// TIA Portal V20 export
DATA_BLOCK "CallEquipment_DB"   // DB155
{ DB_Accessible_From_OPC_UA := 'FALSE' }
// stored: AssignedProDiagFB Unit1.Em2.ProDiag, DBAccessibleFromOPCUA false, DBAccessibleFromWebserver false, InstanceOfName Unit1.Em2.CallEquipment, InstanceOfType FB, Namespace Unit1.Em2
"Unit1.Em2.CallEquipment"
   // VAR_INPUT
   //    ZoneOperationEnable { ExternalWritable := 'False'} : "LWONIK_typeSafetyZoneManualOperation";
   //    unitEnableControlInterfaces { ExternalWritable := 'False'} : "LAF_typeEnableControlInterfaces";
   //    commandExcute { ExternalWritable := 'False'} : Bool;
   // END_VAR
   // VAR_IN_OUT
   //    unitStatus : "LAF_typeUnitStatus";
   //    emFeedback : "LUC_typeEmFeedback";
   //    unitAlarmDB : "LAF_typeAlarms";
   // END_VAR
   // VAR
   //    instSequenceSemiAutoSplice { ExternalWritable := 'False'} : "Unit1.Em2.Sequence_1_SemiAutoSplice";
   //    instTapeUnitInitializedJob1 { ExternalWritable := 'False'} : "LAF_SelectJob";
   //    instAutoSplicerModuleInitializedJob2 { ExternalWritable := 'False'} : "LAF_SelectJob";
   //    instLeftSplicingModuleMoverInitializedJob3 { ExternalWritable := 'False'} : "LAF_SelectJob";
   //    instRightSplicingModuleMoverInitializedJob4 { ExternalWritable := 'False'} : "LAF_SelectJob";
   //    instSplicingModuleMoverAutoJob5 { ExternalWritable := 'False'} : "LAF_SelectJob";
   //    instVacuumAutoJob7 { ExternalWritable := 'False'} : "LAF_SelectJob";
   //    instCutterAutoJob8 { ExternalWritable := 'False'} : "LAF_SelectJob";
   //    instLeftElectrodeReMoverAutoJob9 { ExternalWritable := 'False'} : "LAF_SelectJob";
   //    instRightElectrodeReMoverAutoJob10 { ExternalWritable := 'False'} : "LAF_SelectJob";
   //    instTapeAttachReadyAutoJob11 { ExternalWritable := 'False'} : "LAF_SelectJob";
   //    instTapeAttachStartAutoJob12 { ExternalWritable := 'False'} : "LAF_SelectJob";
   //    instTapeAttachFinishAutoJob13 { ExternalWritable := 'False'} : "LAF_SelectJob";
   //    instLeftSplicingModuleMoverAutoJob14 { ExternalWritable := 'False'} : "LAF_SelectJob";
   //    instRightSplicingModuleMoverAutoJob15 { ExternalWritable := 'False'} : "LAF_SelectJob";
   //    instSemiAutoSpliceFullAutoJob20 { ExternalWritable := 'False'} : "LAF_SelectJob";
   //    instElectrodeFixRightTopFwdBwd { ExternalWritable := 'False'} : "LBC_TwoWayActuatorCn";
   //    instElectrodeFixRightBottomFwdBwd { ExternalWritable := 'False'} : "LBC_TwoWayActuatorCn";
   //    instElectrodeFixLeftTopFwdBwd { ExternalWritable := 'False'} : "LBC_TwoWayActuatorCn";
   //    instElectrodeFixLeftBottomFwdBwd { ExternalWritable := 'False'} : "LBC_TwoWayActuatorCn";
   //    instElectrodeFixLeftTopUpDown { ExternalWritable := 'False'} : "LBC_TwoWayActuatorCn";
   //    instElectrodeFixLeftBottomUpDown { ExternalWritable := 'False'} : "LBC_TwoWayActuatorCn";
   //    instUwSemiSplicerVacuumRightTopOnOff { ExternalWritable := 'False'} : "LBC_TwoWayActuatorCn";
   //    instUwSemiSplicerVacuumRightBottomOnOff { ExternalWritable := 'False'} : "LBC_TwoWayActuatorCn";
   //    instUwSemiSplicerVacuumLeftTopOnOff { ExternalWritable := 'False'} : "LBC_TwoWayActuatorCn";
   //    instUwSemiSplicerVacuumLeftBottomOnOff { ExternalWritable := 'False'} : "LBC_TwoWayActuatorCn";
   //    instElectrodeCutterFwdBwd { ExternalWritable := 'False'} : "LBC_TwoWayActuatorCn";
   //    instSplicingLeftModuleMoverFwdBwd { ExternalWritable := 'False'} : "LBC_TwoWayActuatorCn";
   //    instSplicingRightModuleMoverFwdBwd { ExternalWritable := 'False'} : "LBC_TwoWayActuatorCn";
   //    instElectrodeLeftHolderMoverFwdBwd { ExternalWritable := 'False'} : "LBC_TwoWayActuatorCn";
   //    instElectrodeRightHolderMoverFwdBwd { ExternalWritable := 'False'} : "LBC_TwoWayActuatorCn";
   //    instTapeLoadingTurnCwCcw { ExternalWritable := 'False'} : "LBC_TwoWayActuatorCn";
   //    instTapeAttachUnitFwdBwd { ExternalWritable := 'False'} : "LBC_TwoWayActuatorCn";
   //    instTapeVacuumOnOff { ExternalWritable := 'False'} : "LBC_TwoWayActuatorCn";
   //    instStopperFwdBwd { ExternalWritable := 'False'} : "LBC_TwoWayActuatorCn";
   //    instSupportUnitTransferFwdBwd { ExternalWritable := 'False'} : "LBC_TwoWayActuatorCn";
   //    instSupportUnitShaftUpDown { ExternalWritable := 'False'} : "LBC_TwoWayActuatorCn";
   //    instFrameCoverFwdBwd { ExternalWritable := 'False'} : "LBC_TwoWayActuatorCn";
   //    statUnitStatus { ExternalWritable := 'False'} : "LAF_typeUnitStatus";
   //    instManageAlarms { ExternalWritable := 'False'} : "LAF_ManageAlarms";
   //    instEventsPFE { S7_SetPoint := 'True'} : "Unit1.Em2.EventsPFE";
   //    JobSummary { ExternalWritable := 'False'} : "LAF_typeJobStatus";
   //    statEnableManualCmds { ExternalWritable := 'False'} : Bool;
   //    statPulse { ExternalWritable := 'False'} : Array[0..99] of Bool;
   //    statTonTimer { ExternalWritable := 'False'} : Array[0..99] of TON_TIME;
   //    statTofTimer { ExternalWritable := 'False'} : Array[0..99] of TOF_TIME;
   //    citi_Ptrig : Array[0..20] of Bool;
   //    citiTon : Array[0..20] of TON_TIME;
   //    citi : Time;
   //    citiTest : Array[0..20] of Bool;
   // END_VAR
BEGIN
END_DATA_BLOCK
